// TIA Portal V17 export
FUNCTION_BLOCK "FB_Safety"   // FB100, SCL
   VAR_INPUT
      EStop_Ch1 : Bool;
      EStop_Ch2 : Bool;
   END_VAR
BEGIN
// E-Stop evaluation with fault exit
   IF "I_EStop_Button" AND #EStop_Ch1 AND #EStop_Ch2 THEN
       "DB_Safety".Safety_OK := TRUE;
   ELSE
       GOTO FAULT_EXIT;
   END_IF;
   RETURN;
   FAULT_EXIT:
   "DB_Safety".Safety_OK := FALSE;
   "DB_Safety".Fault_Latch := TRUE;
END_FUNCTION_BLOCK

ORGANIZATION_BLOCK "Main"   // OB1, LAD
BEGIN

REGION Network 1: Call motor control
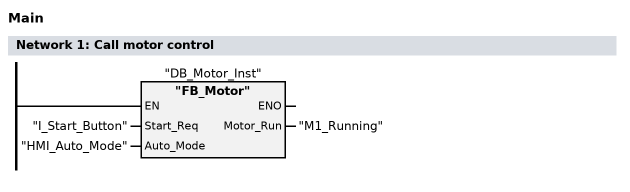
   RUNG wire#powerrail
      "DB_Motor_Inst"(Start_Req := "I_Start_Button", Auto_Mode := "HMI_Auto_Mode", Motor_Run => "M1_Running")
   END_RUNG
   // the same network as SCL:
   "DB_Motor_Inst"(Start_Req := "I_Start_Button", Auto_Mode := "HMI_Auto_Mode", Motor_Run => "M1_Running");   // "FB_Motor"
END_REGION
END_ORGANIZATION_BLOCK
